// TIA Portal V21 export
FUNCTION "DoFc" : Void   // FC109, LAD
{ S7_Optimized_Access := 'FALSE' }
// stored: AutoNumber false, SetENOAutomatically false
   VAR_TEMP   // added for the SCL form of the ladder/FBD networks
      _w1 : Bool;
   END_VAR
BEGIN

REGION Network 2: "DoDb"
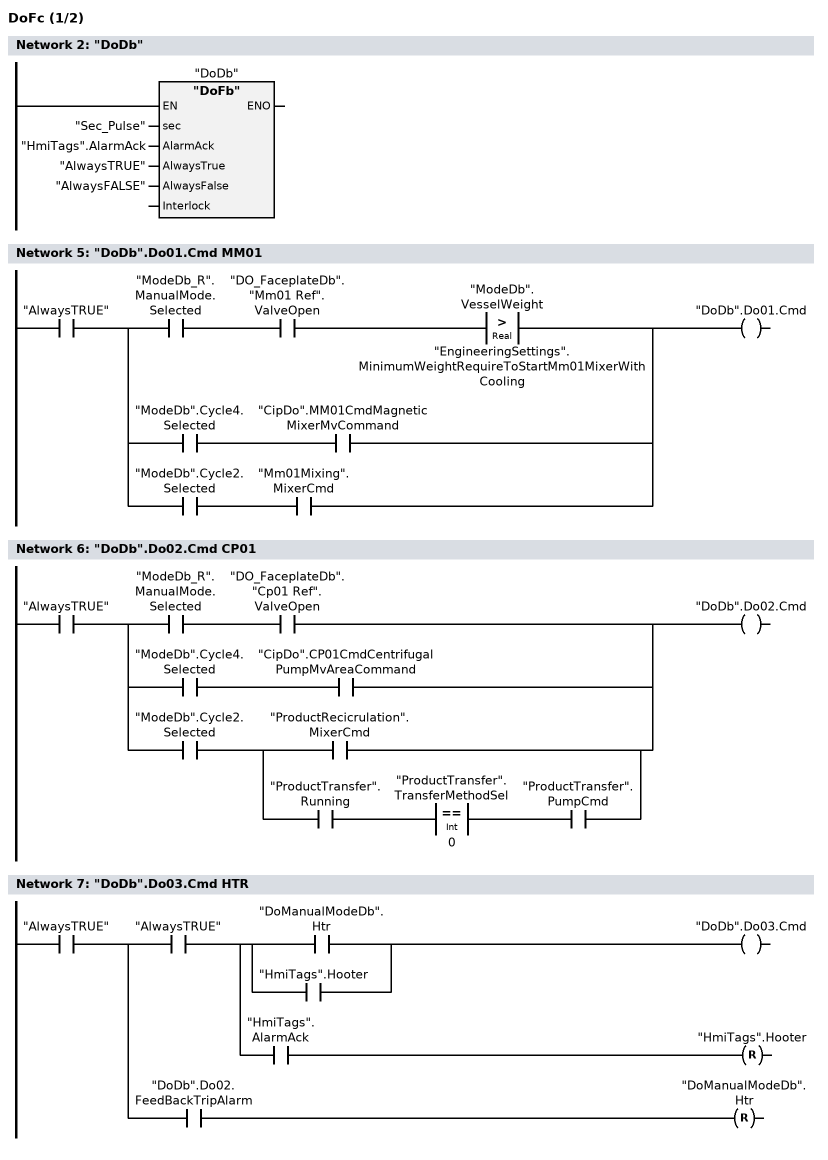
   RUNG wire#powerrail
      "DoDb"(sec := "Sec_Pulse", AlarmAck := "HmiTags".AlarmAck, AlwaysTrue := "AlwaysTRUE", AlwaysFalse := "AlwaysFALSE", Interlock :=)
   END_RUNG
   // the same network as SCL:
   "DoDb"(sec := "Sec_Pulse",   // "DoFb"
          AlarmAck := "HmiTags".AlarmAck,
          AlwaysTrue := "AlwaysTRUE",
          AlwaysFalse := "AlwaysFALSE");
END_REGION

REGION Network 3 (SCL): Digital Output
   "Mm01Cmd":= "DoDb".Do01."Output";
   "Cp01Cmd" := "DoDb".Do02."Output";
   "Htr" := "DoDb".Do03."Output" OR "DoDb".Do03.Cmd;
   "Lf01" := "DoDb".Do04."Output" OR "DoDb".Do04.Cmd;
   "DoSpare1" := "DoDb".Do05."Output";
   "DoSpare2" := "DoDb".Do06."Output";
   "DoSpare3" := "DoDb".Do07."Output";
   "DoSpare4" := "DoDb".Do08."Output";
   "DoSpare5" := "DoDb".Do09."Output";
   "DoSpare6" := "DoDb".Do10."Output";
END_REGION

REGION Network 4 (SCL): MANUAL MODE SELECTED
   //"DoDb".Do01.ManualModeSelected := "ModeDb".MV5000.Mode.ManualMode.Selected;
   "DoDb".Do01.ModeSel := "ModeDb_R".ManualMode.Selected;
   "DoDb".Do02.ModeSel := "ModeDb_R".ManualMode.Selected;
   "DoDb".Do03.ModeSel := "ModeDb_R".ManualMode.Selected;
   "DoDb".Do04.ModeSel := "ModeDb_R".ManualMode.Selected;
   "DoDb".Do05.ModeSel := "ModeDb_R".ManualMode.Selected;
END_REGION

REGION Network 5: "DoDb".Do01.Cmd MM01
   RUNG wire#powerrail
      Contact( "AlwaysTRUE" )
      wire#w1
      Contact( "ModeDb_R".ManualMode.Selected )
      Contact( "DO_FaceplateDb"."Mm01 Ref".ValveOpen )
      { S7_Templates := "SrcType := Real" } GT_Contact(in1 := "ModeDb".VesselWeight, in2 := "EngineeringSettings".MinimumWeightRequireToStartMm01MixerWithCooling)
      wire#w2
      Coil( "DoDb".Do01.Cmd )
   END_RUNG
   RUNG wire#w1
      Contact( "ModeDb".Cycle4.Selected )
      Contact( "CipDo".MM01CmdMagneticMixerMvCommand )
   END_RUNG wire#w2
   RUNG wire#w1
      Contact( "ModeDb".Cycle2.Selected )
      Contact( "Mm01Mixing".MixerCmd )
   END_RUNG wire#w2
   // the same network as SCL:
   "DoDb".Do01.Cmd := "AlwaysTRUE" AND (("ModeDb_R".ManualMode.Selected AND "DO_FaceplateDb"."Mm01 Ref".ValveOpen AND ("ModeDb".VesselWeight > "EngineeringSettings".MinimumWeightRequireToStartMm01MixerWithCooling)) OR ("ModeDb".Cycle4.Selected AND "CipDo".MM01CmdMagneticMixerMvCommand) OR ("ModeDb".Cycle2.Selected AND "Mm01Mixing".MixerCmd));
END_REGION

REGION Network 6: "DoDb".Do02.Cmd CP01
   RUNG wire#powerrail
      Contact( "AlwaysTRUE" )
      wire#w1
      Contact( "ModeDb_R".ManualMode.Selected )
      Contact( "DO_FaceplateDb"."Cp01 Ref".ValveOpen )
      wire#w2
      Coil( "DoDb".Do02.Cmd )
   END_RUNG
   RUNG wire#w1
      Contact( "ModeDb".Cycle4.Selected )
      Contact( "CipDo".CP01CmdCentrifugalPumpMvAreaCommand )
   END_RUNG wire#w2
   RUNG wire#w1
      Contact( "ModeDb".Cycle2.Selected )
      wire#w3
      Contact( "ProductRecicrulation".MixerCmd )
   END_RUNG wire#w2
   RUNG wire#w3
      Contact( "ProductTransfer".Running )
      { S7_Templates := "SrcType := Int" } EQ_Contact(in1 := "ProductTransfer".TransferMethodSel, in2 := 0)
      Contact( "ProductTransfer".PumpCmd )
   END_RUNG wire#w2
   // the same network as SCL:
   "DoDb".Do02.Cmd := "AlwaysTRUE" AND (("ModeDb_R".ManualMode.Selected AND "DO_FaceplateDb"."Cp01 Ref".ValveOpen) OR ("ModeDb".Cycle4.Selected AND "CipDo".CP01CmdCentrifugalPumpMvAreaCommand) OR ("ModeDb".Cycle2.Selected AND ("ProductRecicrulation".MixerCmd OR ("ProductTransfer".Running AND ("ProductTransfer".TransferMethodSel = 0) AND "ProductTransfer".PumpCmd))));
END_REGION

REGION Network 7: "DoDb".Do03.Cmd HTR
   RUNG wire#powerrail
      Contact( "AlwaysTRUE" )
      wire#w1
      Contact( "AlwaysTRUE" )
      wire#w2
      Contact( "DoManualModeDb".Htr )
      wire#w3
      Coil( "DoDb".Do03.Cmd )
   END_RUNG
   RUNG wire#w2
      Contact( "HmiTags".Hooter )
   END_RUNG wire#w3
   RUNG wire#w2
      Contact( "HmiTags".AlarmAck )
      R_Coil( "HmiTags".Hooter )
   END_RUNG
   RUNG wire#w1
      Contact( "DoDb".Do02.FeedBackTripAlarm )
      R_Coil( "DoManualModeDb".Htr )
   END_RUNG
   // the same network as SCL:
   #_w1 := "AlwaysTRUE" AND "AlwaysTRUE";
   "DoDb".Do03.Cmd := #_w1 AND ("DoManualModeDb".Htr OR "HmiTags".Hooter);
   IF #_w1 AND "HmiTags".AlarmAck THEN "HmiTags".Hooter := FALSE; END_IF;
   IF "AlwaysTRUE" AND "DoDb".Do02.FeedBackTripAlarm THEN "DoManualModeDb".Htr := FALSE; END_IF;
END_REGION

REGION Network 8: "DoDb".Do04.Cmd
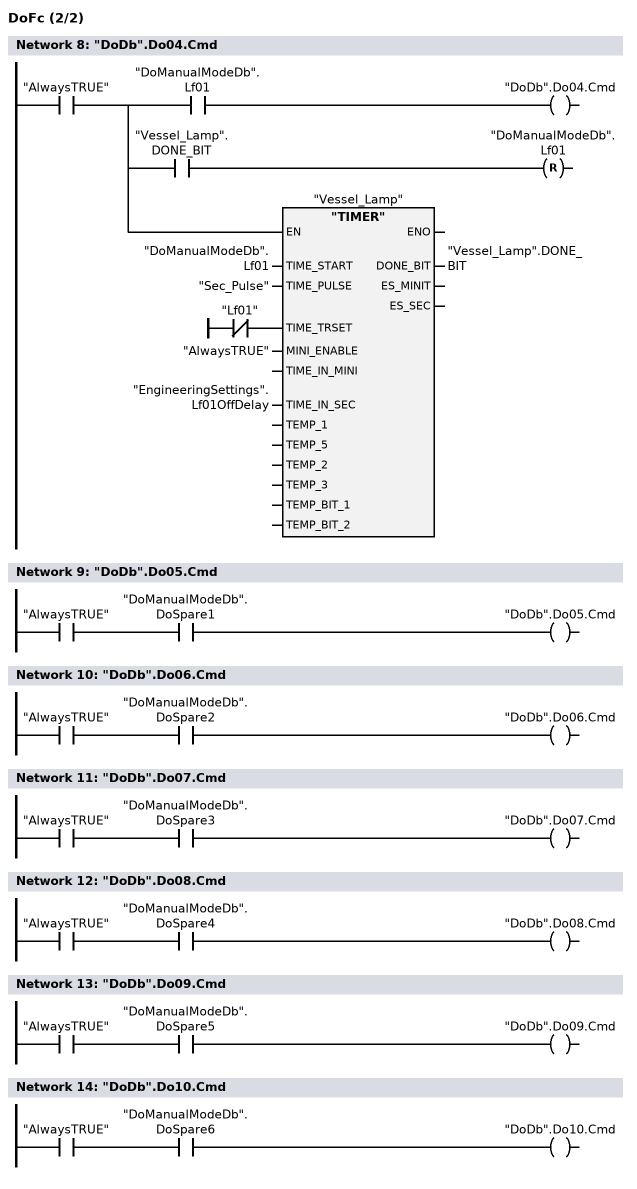
   RUNG wire#powerrail
      Contact( "AlwaysTRUE" )
      wire#w1
      Contact( "DoManualModeDb".Lf01 )
      Coil( "DoDb".Do04.Cmd )
   END_RUNG
   RUNG wire#w1
      Contact( "Vessel_Lamp".DONE_BIT )
      R_Coil( "DoManualModeDb".Lf01 )
   END_RUNG
   RUNG wire#w1
      "Vessel_Lamp"(TIME_TRSET := wire#w2, TIME_START := "DoManualModeDb".Lf01, TIME_PULSE := "Sec_Pulse", MINI_ENABLE := "AlwaysTRUE", TIME_IN_MINI :=, TIME_IN_SEC := "EngineeringSettings".Lf01OffDelay, TEMP_1 :=, TEMP_5 :=, TEMP_2 :=, TEMP_3 :=, TEMP_BIT_1 :=, TEMP_BIT_2 :=, DONE_BIT => "Vessel_Lamp".DONE_BIT, ES_MINIT =>, ES_SEC =>)
   END_RUNG
   RUNG wire#powerrail
      I_Contact( "Lf01" )
   END_RUNG wire#w2
   // the same network as SCL:
   "DoDb".Do04.Cmd := "AlwaysTRUE" AND "DoManualModeDb".Lf01;
   IF "AlwaysTRUE" AND "Vessel_Lamp".DONE_BIT THEN "DoManualModeDb".Lf01 := FALSE; END_IF;
   IF "AlwaysTRUE" THEN
       "Vessel_Lamp"(TIME_START := "DoManualModeDb".Lf01,   // "TIMER"
                     TIME_PULSE := "Sec_Pulse",
                     TIME_TRSET := NOT "Lf01",
                     MINI_ENABLE := "AlwaysTRUE",
                     TIME_IN_SEC := "EngineeringSettings".Lf01OffDelay,
                     DONE_BIT => "Vessel_Lamp".DONE_BIT);
   END_IF;
END_REGION

REGION Network 9: "DoDb".Do05.Cmd
   RUNG wire#powerrail
      Contact( "AlwaysTRUE" )
      Contact( "DoManualModeDb".DoSpare1 )
      Coil( "DoDb".Do05.Cmd )
   END_RUNG
   // the same network as SCL:
   "DoDb".Do05.Cmd := "AlwaysTRUE" AND "DoManualModeDb".DoSpare1;
END_REGION

REGION Network 10: "DoDb".Do06.Cmd
   RUNG wire#powerrail
      Contact( "AlwaysTRUE" )
      Contact( "DoManualModeDb".DoSpare2 )
      Coil( "DoDb".Do06.Cmd )
   END_RUNG
   // the same network as SCL:
   "DoDb".Do06.Cmd := "AlwaysTRUE" AND "DoManualModeDb".DoSpare2;
END_REGION

REGION Network 11: "DoDb".Do07.Cmd
   RUNG wire#powerrail
      Contact( "AlwaysTRUE" )
      Contact( "DoManualModeDb".DoSpare3 )
      Coil( "DoDb".Do07.Cmd )
   END_RUNG
   // the same network as SCL:
   "DoDb".Do07.Cmd := "AlwaysTRUE" AND "DoManualModeDb".DoSpare3;
END_REGION

REGION Network 12: "DoDb".Do08.Cmd
   RUNG wire#powerrail
      Contact( "AlwaysTRUE" )
      Contact( "DoManualModeDb".DoSpare4 )
      Coil( "DoDb".Do08.Cmd )
   END_RUNG
   // the same network as SCL:
   "DoDb".Do08.Cmd := "AlwaysTRUE" AND "DoManualModeDb".DoSpare4;
END_REGION

REGION Network 13: "DoDb".Do09.Cmd
   RUNG wire#powerrail
      Contact( "AlwaysTRUE" )
      Contact( "DoManualModeDb".DoSpare5 )
      Coil( "DoDb".Do09.Cmd )
   END_RUNG
   // the same network as SCL:
   "DoDb".Do09.Cmd := "AlwaysTRUE" AND "DoManualModeDb".DoSpare5;
END_REGION

REGION Network 14: "DoDb".Do10.Cmd
   RUNG wire#powerrail
      Contact( "AlwaysTRUE" )
      Contact( "DoManualModeDb".DoSpare6 )
      Coil( "DoDb".Do10.Cmd )
   END_RUNG
   // the same network as SCL:
   "DoDb".Do10.Cmd := "AlwaysTRUE" AND "DoManualModeDb".DoSpare6;
END_REGION

REGION Network 15 (SCL): Fb delay
   "DoDb".Do01.FBCheckDelay := "EngineeringSettings"."Mm01F/BDelay";
   "DoDb".Do02.FBCheckDelay := "EngineeringSettings"."Cp01F/BDelay";
   //"VesselLamp_DB".LF01.TIME_IN_SEC := "EngineeringSettings".Lf01OffDelay;
END_REGION

REGION Network 16 (SCL): FeedBack Alarms And Input
   "DoDb".Do01.MotorFeedbackInputSelection := 1;
   "DoDb".Do02.MotorFeedbackInputSelection := 1;

   "DoDb".Do01.MotorFeedbackInput := "DiFinal".MagneticMixerFeedback;
   "DoDb".Do02.MotorFeedbackInput := "DiFinal".CipPumpFeedback;

   "DoDb".Do02.FeedBackTripAlarm := "SafetyAlarms".Cp01FeedbackTrip;
   "DoDb".Do01.FeedBackTripAlarm := "SafetyAlarms".Mm01FeedbackTrip;


   "SafetyAlarms".Mm01FeedbackTrip := "DoDb".Do01.FeedBackTripAlarm;
   "SafetyAlarms".Cp01FeedbackTrip := "DoDb".Do02.FeedBackTripAlarm;

   "SafetyAlarms".Mm01FeedbackTrip := "DoDb".Do01.OpFbTrip;
   "SafetyAlarms".Cp01FeedbackTrip := "DoDb".Do02.OpFbTrip;

   "DoDb".Do01.AlarmAck := "HmiTags".AlarmAck;
   "DoDb".Do02.AlarmAck := "HmiTags".AlarmAck;
END_REGION
END_FUNCTION
